Staubli VAL3: printList.pgx

program printList(num x_nType (dimensions=1))
  local num i
  local num l_nX
  local string l_sProg
  local num l_nIndex
  local num l_nSize[3]
  local num l_nDone
  local num l_nTotal
  local num l_nZero
begin
  //
  l_nZero=0
  call use:getListPosition(l_nX,l_nZero)
  // get the size
  call processList:getSize(l_nSize,x_nType)
  // resize it
  if l_nSize!=0
    l_nSize=l_nSize-1
  endIf
  // print the process start LIST
  for i=cycleStatus:nProg to min(l_nSize-cycleStatus:nProg,1)
    call processList:getCycle(l_sProg,l_nTotal,l_nDone,i,x_nType)
    if l_sProg!=""
      if i==cycleStatus:nProg
        setTextMode(1)
      endIf
      call use:strfill(l_sProg,10,l_sProg)
      l_sProg=l_sProg+"["+toString("1",l_nDone)+"/"+toString("1",l_nTotal)+"]"
      call use:type(0,i+1,l_sProg)
      setTextMode(0)
      call use:typeLen(len(l_sProg),i+1,"",l_nX-1-len(l_sProg))
      l_nIndex=l_nIndex+1
    endIf
  endFor
  // write the empty space
  if l_nIndex<2
    for i=l_nIndex to 1
      // empty Line
      call use:typeLen(0,i+1,"",l_nX-1)
    endFor
  endIf
end
